{attribute 'qualified_only'}
{attribute 'strict'}
{attribute 'to_string'}
TYPE ST120_Cylinders_e :
(
    GreiferLinks,
    GreiferRechts,
	SchwenkenLinks,
	SchwenkenRechts,
	HubladerLinks,
	HubladerRechts,
    _max
);
END_TYPE

(* stored: Version 1.1.0.1, ProductVersion 3.1.4024.6
   EnumerationTextList ST120_Cylinders_e: Id {30c20dce-e666-4402-bb4e-c41ede9fdffa} *)
